ORGANIZATION_BLOCK MAIN:OB1
TITLE=HSC Test Program
BEGIN
Network 1
LD     SM0.1
MOVB   0, VB100
MOVW   0, VW100
MOVW   0, VW102

Network 2
LD     SM0.1
MOVB   16#F8, SMB37
MOVW   0, SMW38
MOVW   0, SMW42
HDEF   0, 0
HSC    0

Network 3
LD     SM0.0
MOVW   SMW38, VW100
MOVW   SMW48, VW102

END_ORGANIZATION_BLOCK
